TYPE stCu_ProcessData EXTENDS stCu_ProcessDataBase : 
STRUCT
    {attribute addProperty Name "A_Check_1"}
    A_Check_1 : fbAnalogueValueData;
    {attribute addProperty Name "A_Check_2"}
    A_Check_2 : fbAnalogueValueData;
    {attribute addProperty Name "A_Check_3"}
    A_Check_3 : fbAnalogueValueData;
    {attribute addProperty Name "A_Check_4"}
    A_Check_4 : fbAnalogueValueData;
    {attribute addProperty Name "A_Check_5"}
    A_Check_5 : fbAnalogueValueData;
    {attribute clr [RenderIgnore("Display", "ShadowDisplay")]}
    {attribute addProperty Name "A_Check_6"}
    A_Check_6 : fbAnalogueValueData;
    {attribute clr [RenderIgnore("Control", "ShadowControl")]}
    {attribute addProperty Name "A_Check_7"}
    A_Check_7 : fbAnalogueValueData;
END_STRUCT
END_TYPE

(* stored: Version 1.1.0.1, ProductVersion 3.1.4024.6
   DUT stCu_ProcessData: Id {c4d175d0-d947-48c0-b915-c3fe6d62b327} *)
